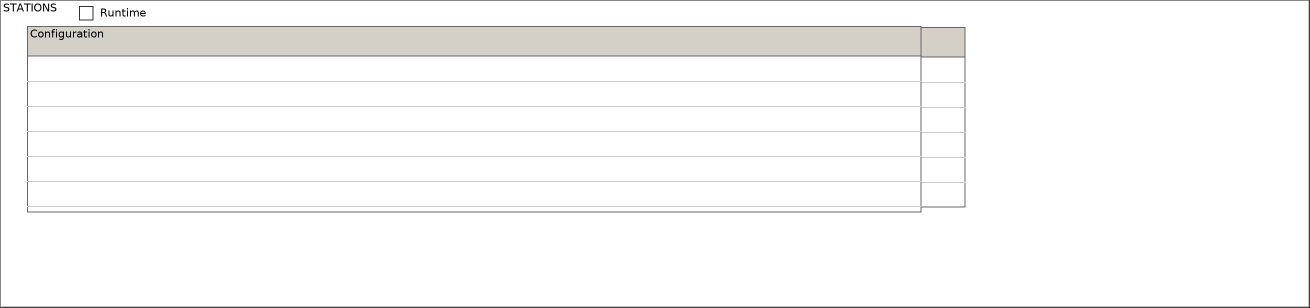
VISUALIZATION VI_StationsVISU  // 1310x308
VAR_IN_OUT
	aStations		: ARRAY [1..Tc3_XTS_Utility.TcIoXtsEnvironmentParameterList.MaxXtsInfoStation] OF FB_Station; //Stations
END_VAR
VAR
	stTableStruct : ARRAY [1..25] OF stTableStructx10;
	iSelectedStation : INT;
	bRunTime		: BOOL;
END_VAR
    Rectangle (0,0 1310x308), "STATIONS"
    Table (27,27 938x180), "Configuration", invisible if: bRunTime=true, data array: stTableStruct
        p1137915858: iSelectedStation
        p3854506369: aStations[INDEX].stCfg.sName
        p1892666644: aStations[INDEX].stCfg.lrStartPosition
        p338671338: aStations[INDEX].stCfg.lrStopPosition[1]
        p2170511999: aStations[INDEX].stCfg.lrStopPosition[2]
        p3723444502: aStations[INDEX].stCfg.lrStopPosition[3]
        p1218418051: aStations[INDEX].stCfg.lrProcessingTime
        p746581629: aStations[INDEX].stCfg.uiNumStopPositions
        p3104783080: aStations[INDEX].stCfg.lrTravelTime
        p7306298: aStations[INDEX].stCfg.lrEndPosition
        p511219082: Start Position
        p1755163831: Stop Position 1
        p4092479075: Stop Position 2
        p2237128397: Stop Position 3
        p505689113: Process Time
        p1757482276: Stop Positions
        p4088588272: Travel Time
        p2243050616: Extra Cfg.
        p516019884: End Position
        p2685023577: stTableStruct.b1
        p3312258591: stTableStruct.b2
        p1791247317: stTableStruct.b3
        p262371475: stTableStruct.b4
        p4008173056: stTableStruct.b5
        p2340480326: stTableStruct.b6
        p606709900: stTableStruct.b7
        p1095668682: stTableStruct.b8
        p1037165547: stTableStruct.b9
        p1488378029: stTableStruct.b10
        Columns.Column.[3].Template: OnMouseClick: write the text variable via Default
        Columns.Column.[6].Template: OnMouseClick: write the text variable via Default, min 1, max 3
        Columns.Column.[4].Template: OnMouseClick: write the text variable via Default
        Columns.Column.[5].Template: OnMouseClick: write the text variable via Default
        Columns.Column.[2].Template: OnMouseClick: write the text variable via Default
        Columns.Column.[7].Template: OnMouseClick: write the text variable via Default
        Columns.Column.[9].Template: OnMouseClick: write the text variable via Default
        Columns.Column.[1].Template: OnMouseClick: write the text variable via Default
    Checkbox (77,2 150x22), "Runtime", variable: bRunTime
    Table (27,26 894x186), "Configuration", invisible if: bRunTime=false, data array: stTableStruct
        p225073791: %5.2f s/m
        p3854506369: aStations[INDEX].stCfg.sName
        p1892666644: aStations[INDEX].stCfg.bEnableManualAck
        p338671338: aStations[INDEX].stCfg.bManualAck
        p2170511999: aStations[INDEX].fbMoversFIFO.nMovers
        p3723444502: aStations[INDEX].stCfg.udiSequenceState
        p1218418051: aStations[INDEX].udiErrorID
        p746581629: aStations[INDEX].sMoversWaiting
        p3104783080: aStations[INDEX].sMoversIn
        p2501879983: (aStations[INDEX].lrActualProcessTime+aStations[INDEX].lrActualWaitingTime)/udint_to_lreal(aStations[INDEX].stCfg.uiNumStopPositions)
        p7306298: xts.aStations[INDEX].lrActualWaitingTime
        p511219082: M. Ack
        p4092479075: Movers Waiting
        p505689113: Error ID
        p4088588272: Movers In
        p2243050616: Cycle Time
        p516019884: Waiting Time
        p2685023577: stTableStruct.b1
        p3312258591: stTableStruct.b2
        p1791247317: stTableStruct.b3
        p262371475: stTableStruct.b4
        p4008173056: stTableStruct.b5
        p2340480326: stTableStruct.b6
        p606709900: stTableStruct.b7
        p1095668682: stTableStruct.b8
        p1037165547: stTableStruct.b9
        p1488378029: stTableStruct.b10
        Columns.Column.[6].Template: OnMouseClick: write the text variable via Default, min 1, max 3
        Columns.Column.[4].Template: OnMouseClick: write the text variable via Default
        Columns.Column.[5].Template: OnMouseClick: write the text variable via Default
        Columns.Column.[2].Template: tap aStations[INDEX].stCfg.bManualAck
        Columns.Column.[0].Template: OnMouseClick: write the text variable via Default
        Columns.Column.[7].Template: OnMouseClick: write the text variable via Default
        Columns.Column.[9].Template: OnMouseClick: write the text variable via Default
        Columns.Column.[1].Template: toggle aStations[INDEX].stCfg.bEnableManualAck
END_VISUALIZATION

(* stored: Version 1.1.0.1, ProductVersion 3.1.4024.11
   Visu VI_StationsVISU: Id {852d93b2-cd24-46f9-bfa8-cc8d837fda15} *)
